TYPE WcStateInputToggleBase_F68C23A9 :
STRUCT
END_STRUCT
END_TYPE

(* stored: Version 1.2.0.0, ProductVersion 3.1.4024.9
   DUT WcStateInputToggleBase_F68C23A9: Id {ab9df3d3-75cb-4417-8524-a5aeb3bd7b1c} *)
